KUKA KRL program: S_11_pc_at_cell_01.src, S_11_pc_at_cell_01.dat

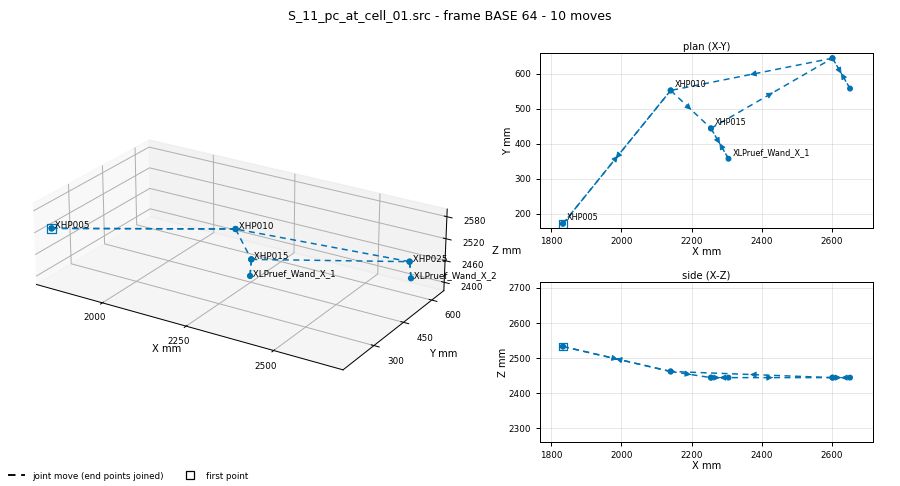
[picture p0: tool path of S_11_pc_at_cell_01.src in frame BASE 64, 10 of 12 moves have a stored position in this frame; points joined in program order, loops and branches not executed]
--- S_11_pc_at_cell_01.src ---
&ACCESS RVP
&REL 9
&COMMENT DAI_H_SOP_pc_at_cell_01
&PARAM EDITMASK = DAI
&PARAM TEMPLATE = C:\KRC\roboter\template\vg_appl
&PARAM DISKPATH = KRC:\R1\H_Prog\DAI_SOP
DEF S_11_pc_at_cell_01( )
;FOLD INI;%{PE}
  ;FOLD BASISTECH INI
    GLOBAL INTERRUPT DECL 3 WHEN $STOPMESS==TRUE DO IR_STOPM ( )
    INTERRUPT ON 3
    BAS (#INITMOV,0 )
  ;ENDFOLD (BASISTECH INI)
  ;FOLD USER INI
    ;Make your modifications here
  ;ENDFOLD (USER INI)
;ENDFOLD (INI)
;FOLD ; Anlagenbezeichn: HC53_C    Stations-Nr: 060RB_100;%{PE}
;FOLD Parameters ;%{h}
;Params IlfProvider=kukaroboter.basistech.inlineforms.comments.comment; Kuka.Content=Anlagenbezeichn: HC53_C    Stations-Nr: 060RB_100
;ENDFOLD
;ENDFOLD
;FOLD ; Stand / Version: V1.0;%{PE}
;FOLD Parameters ;%{h}
;Params IlfProvider=kukaroboter.basistech.inlineforms.comments.comment; Kuka.Content=Stand / Version: V1.0
;ENDFOLD
;ENDFOLD
;FOLD ; Name Bearbeiter: EBZ-AE;%{PE}
;FOLD Parameters ;%{h}
;Params IlfProvider=kukaroboter.basistech.inlineforms.comments.comment; Kuka.Content=Name Bearbeiter: EBZ-AE
;ENDFOLD
;ENDFOLD
;FOLD ; Translator Version:29.01.2024 - Version 15.08;%{PE}
;FOLD Parameters ;%{h}
;Params IlfProvider=kukaroboter.basistech.inlineforms.comments.comment; Kuka.Content=Translator Version:29.01.2024 - Version 15.08
;ENDFOLD
;ENDFOLD

REPEAT

;FOLD MSG_T1
MSG_SHOW("DAI_H_SOP",#quit,999,"dai_h_sop_ok_0")
;ENDFOLD

; ***************************************
; A C H T U N G !!! Nur in $T1 abfahren
; ***************************************
UNTIL $T1 == TRUE

; ***************************************
; Pruefende Waende = 2
;----------------------------------------
; Lademagazin in undefinierte
; Position verfahren, damit Raum
; aktiviert wird.
;FOLD WAIT FOR ( IN 1026 'Vordefinierter Eingang immer ruckgesetzt.' )  ;%{PE}
;FOLD Parameters ;%{h}
;Params IlfProvider=kukaroboter.basistech.inlineforms.logics.waitfor; Kuka.WaitLogicTerm1=None; Kuka.WaitForNot1=False; Kuka.WaitLogicOp2.Term1=None; Kuka.WaitForNot2.Term1=False; Kuka.WaitForSysVar2.Term1=IN; Kuka.WaitForIndex2.Term1=1026; Kuka.WaitForIndexName2.Term1=Vordefinierter Eingang immer ruckgesetzt.; Kuka.WaitForTermNumbers=1; Kuka.WaitForOpNumbers=2; Kuka.WaitForCont=False
;ENDFOLD
WAIT FOR  ( $IN[1026] )
;ENDFOLD
; ***************************************

;FOLD PTP HOME Vel=100 % DEFAULT;%{PE}
;FOLD Parameters ;%{h}
;Params IlfProvider=kukaroboter.basistech.inlineforms.movement.old; Kuka.IsGlobalPoint=False; Kuka.PointName=HOME; Kuka.BlendingEnabled=False; Kuka.MoveDataPtpName=DEFAULT; Kuka.VelocityPtp=100; Kuka.CurrentCDSetIndex=0; Kuka.MovementParameterFieldEnabled=True; IlfCommand=PTP
;ENDFOLD
$BWDSTART = FALSE
PDAT_ACT = PDEFAULT
FDAT_ACT = FHOME
BAS(#PTP_PARAMS, 100.0)
SET_CD_PARAMS (0)
PTP XHOME
;ENDFOLD

;Dynamische Pruefung Teil vorhanden
;FOLD PartPresent.CheckOff #1:5277, #2:5278, #3:1025, #4:1025, #5:1025, #6:1025, Bounce Time:100, Constant: Yes;%{PE}%
CheckPartPresent(5277,5278,1025,1025,1025,1025,100, True,FALSE)
;ENDFOLD

;Greifer-Ventile betatigen/pruefen
;FOLD DAI_GripValveCheck.Valve2 State:Fixierstift Ausfahren Gs, 060GRH101-QM1;%{PE}%
CheckValveState(2,1)
;ENDFOLD
;FOLD DAI_GripValveCheck.Valve3 State:Spanner Oeffnen Gs, 060GRH101-QM2;%{PE}%
CheckValveState(3,1)
;ENDFOLD
;FOLD DAI_GripValveCheck.Valve4 State:Spanner Oeffnen Gs, 060GRH101-QM3;%{PE}%
CheckValveState(4,1)
;ENDFOLD

;FOLD PTP HP005 Vel=100 % PDAT2 Tool[64]:Zero Base[64]:Zero;%{PE}
;FOLD Parameters ;%{h}
;Params IlfProvider=kukaroboter.basistech.inlineforms.movement.old; Kuka.IsGlobalPoint=False; Kuka.PointName=HP005; Kuka.BlendingEnabled=False; Kuka.MoveDataPtpName=PDAT2; Kuka.VelocityPtp=100; Kuka.CurrentCDSetIndex=0; Kuka.MovementParameterFieldEnabled=True; IlfCommand=PTP
;ENDFOLD
$BWDSTART = FALSE
PDAT_ACT = PPDAT2
FDAT_ACT = FHP005
BAS(#PTP_PARAMS, 100.0)
SET_CD_PARAMS (0)
PTP XHP005
;ENDFOLD
;FOLD PTP HP010 Vel=100 % PDAT3 Tool[64]:Zero Base[64]:Zero;%{PE}
;FOLD Parameters ;%{h}
;Params IlfProvider=kukaroboter.basistech.inlineforms.movement.old; Kuka.IsGlobalPoint=False; Kuka.PointName=HP010; Kuka.BlendingEnabled=False; Kuka.MoveDataPtpName=PDAT3; Kuka.VelocityPtp=100; Kuka.CurrentCDSetIndex=0; Kuka.MovementParameterFieldEnabled=True; IlfCommand=PTP
;ENDFOLD
$BWDSTART = FALSE
PDAT_ACT = PPDAT3
FDAT_ACT = FHP010
BAS(#PTP_PARAMS, 100.0)
SET_CD_PARAMS (0)
PTP XHP010
;ENDFOLD
;FOLD PTP HP015 Vel=100 % PDAT4 Tool[64]:Zero Base[64]:Zero;%{PE}
;FOLD Parameters ;%{h}
;Params IlfProvider=kukaroboter.basistech.inlineforms.movement.old; Kuka.IsGlobalPoint=False; Kuka.PointName=HP015; Kuka.BlendingEnabled=False; Kuka.MoveDataPtpName=PDAT4; Kuka.VelocityPtp=100; Kuka.CurrentCDSetIndex=0; Kuka.MovementParameterFieldEnabled=True; IlfCommand=PTP
;ENDFOLD
$BWDSTART = FALSE
PDAT_ACT = PPDAT4
FDAT_ACT = FHP015
BAS(#PTP_PARAMS, 100.0)
SET_CD_PARAMS (0)
PTP XHP015
;ENDFOLD

; Pruefung Flache 1 erste Position
;FOLD PTP LPruef_Wand_X_1 Vel=100 % PDAT04 Tool[64]:Zero Base[64]:Zero ;%{PE}
;FOLD Parameters ;%{h}
;Params IlfProvider=kukaroboter.basistech.inlineforms.movement.old; Kuka.IsGlobalPoint=False; Kuka.PointName=LPruef_Wand_X_1; Kuka.BlendingEnabled=False; Kuka.MoveDataPtpName=PDAT04; Kuka.VelocityPtp=100; Kuka.CurrentCDSetIndex=0; Kuka.MovementParameterFieldEnabled=True; IlfCommand=PTP
;ENDFOLD
$BWDSTART = FALSE
PDAT_ACT = PPDAT04
FDAT_ACT = FLPruef_Wand_X_1
BAS(#PTP_PARAMS, 100.0)
SET_CD_PARAMS (0)
PTP XLPruef_Wand_X_1
;ENDFOLD

;FOLD PTP HP020 Vel=100 % PDAT03 Tool[64]:Zero Base[64]:Zero ;%{PE}
;FOLD Parameters ;%{h}
;Params IlfProvider=kukaroboter.basistech.inlineforms.movement.old; Kuka.IsGlobalPoint=False; Kuka.PointName=HP020; Kuka.BlendingEnabled=False; Kuka.MoveDataPtpName=PDAT03; Kuka.VelocityPtp=100; Kuka.CurrentCDSetIndex=0; Kuka.MovementParameterFieldEnabled=True; IlfCommand=PTP
;ENDFOLD
$BWDSTART = FALSE
PDAT_ACT = PPDAT03
FDAT_ACT = FHP020
BAS(#PTP_PARAMS, 100.0)
SET_CD_PARAMS (0)
PTP XHP020
;ENDFOLD

;FOLD PTP HP025 Vel=100 % PDAT7 Tool[64]:Zero Base[64]:Zero;%{PE}
;FOLD Parameters ;%{h}
;Params IlfProvider=kukaroboter.basistech.inlineforms.movement.old; Kuka.IsGlobalPoint=False; Kuka.PointName=HP025; Kuka.BlendingEnabled=False; Kuka.MoveDataPtpName=PDAT7; Kuka.VelocityPtp=100; Kuka.CurrentCDSetIndex=0; Kuka.MovementParameterFieldEnabled=True; IlfCommand=PTP
;ENDFOLD
$BWDSTART = FALSE
PDAT_ACT = PPDAT7
FDAT_ACT = FHP025
BAS(#PTP_PARAMS, 100.0)
SET_CD_PARAMS (0)
PTP XHP025
;ENDFOLD

; Pruefung Flache 1 zweite Position
;FOLD PTP LPruef_Wand_X_2 Vel=100 % PDAT02 Tool[64]:Zero Base[64]:Zero ;%{PE}
;FOLD Parameters ;%{h}
;Params IlfProvider=kukaroboter.basistech.inlineforms.movement.old; Kuka.IsGlobalPoint=False; Kuka.PointName=LPruef_Wand_X_2; Kuka.BlendingEnabled=False; Kuka.MoveDataPtpName=PDAT02; Kuka.VelocityPtp=100; Kuka.CurrentCDSetIndex=0; Kuka.MovementParameterFieldEnabled=True; IlfCommand=PTP
;ENDFOLD
$BWDSTART = FALSE
PDAT_ACT = PPDAT02
FDAT_ACT = FLPruef_Wand_X_2
BAS(#PTP_PARAMS, 100.0)
SET_CD_PARAMS (0)
PTP XLPruef_Wand_X_2
;ENDFOLD

;FOLD PTP HP030 Vel=100 % PDAT01 Tool[64]:Zero Base[64]:Zero ;%{PE}
;FOLD Parameters ;%{h}
;Params IlfProvider=kukaroboter.basistech.inlineforms.movement.old; Kuka.IsGlobalPoint=False; Kuka.PointName=HP030; Kuka.BlendingEnabled=False; Kuka.MoveDataPtpName=PDAT01; Kuka.VelocityPtp=100; Kuka.CurrentCDSetIndex=0; Kuka.MovementParameterFieldEnabled=True; IlfCommand=PTP
;ENDFOLD
$BWDSTART = FALSE
PDAT_ACT = PPDAT01
FDAT_ACT = FHP030
BAS(#PTP_PARAMS, 100.0)
SET_CD_PARAMS (0)
PTP XHP030
;ENDFOLD

;FOLD PTP HP040 Vel=100 % PDAT05 Tool[64]:Zero Base[64]:Zero ;%{PE}
;FOLD Parameters ;%{h}
;Params IlfProvider=kukaroboter.basistech.inlineforms.movement.old; Kuka.IsGlobalPoint=False; Kuka.PointName=HP040; Kuka.BlendingEnabled=False; Kuka.MoveDataPtpName=PDAT05; Kuka.VelocityPtp=100; Kuka.CurrentCDSetIndex=0; Kuka.MovementParameterFieldEnabled=True; IlfCommand=PTP
;ENDFOLD
$BWDSTART = FALSE
PDAT_ACT = PPDAT05
FDAT_ACT = FHP040
BAS(#PTP_PARAMS, 100.0)
SET_CD_PARAMS (0)
PTP XHP040
;ENDFOLD
;FOLD PTP HP045 Vel=100 % PDAT13 Tool[64]:Zero Base[64]:Zero;%{PE}
;FOLD Parameters ;%{h}
;Params IlfProvider=kukaroboter.basistech.inlineforms.movement.old; Kuka.IsGlobalPoint=False; Kuka.PointName=HP045; Kuka.BlendingEnabled=False; Kuka.MoveDataPtpName=PDAT13; Kuka.VelocityPtp=100; Kuka.CurrentCDSetIndex=0; Kuka.MovementParameterFieldEnabled=True; IlfCommand=PTP
;ENDFOLD
$BWDSTART = FALSE
PDAT_ACT = PPDAT13
FDAT_ACT = FHP045
BAS(#PTP_PARAMS, 100.0)
SET_CD_PARAMS (0)
PTP XHP045
;ENDFOLD

;FOLD PTP HOME Vel=100 % DEFAULT;%{PE}
;FOLD Parameters ;%{h}
;Params IlfProvider=kukaroboter.basistech.inlineforms.movement.old; Kuka.IsGlobalPoint=False; Kuka.PointName=HOME; Kuka.BlendingEnabled=False; Kuka.MoveDataPtpName=DEFAULT; Kuka.VelocityPtp=100; Kuka.CurrentCDSetIndex=0; Kuka.MovementParameterFieldEnabled=True; IlfCommand=PTP
;ENDFOLD
$BWDSTART = FALSE
PDAT_ACT = PDEFAULT
FDAT_ACT = FHOME
BAS(#PTP_PARAMS, 100.0)
SET_CD_PARAMS (0)
PTP XHOME
;ENDFOLD

;----------------------------------------
; Lademagazin schliessen und
; und Quittieren.
;FOLD WAIT FOR ( IN 1026 'Vordefinierter Eingang immer ruckgesetzt.' )  ;%{PE}
;FOLD Parameters ;%{h}
;Params IlfProvider=kukaroboter.basistech.inlineforms.logics.waitfor; Kuka.WaitLogicTerm1=None; Kuka.WaitForNot1=False; Kuka.WaitLogicOp2.Term1=None; Kuka.WaitForNot2.Term1=False; Kuka.WaitForSysVar2.Term1=IN; Kuka.WaitForIndex2.Term1=1026; Kuka.WaitForIndexName2.Term1=Vordefinierter Eingang immer ruckgesetzt.; Kuka.WaitForTermNumbers=1; Kuka.WaitForOpNumbers=2; Kuka.WaitForCont=False
;ENDFOLD
WAIT FOR  ( $IN[1026] )
;ENDFOLD
; ***************************************
 ;Collision detection - Off
;FOLD COLLDETECT Off ;%{PE}
;FOLD Parameters ;%{h}
;Params IlfProvider=kukaroboter.basistech.inlineforms.colldetect.off; CollDetect.Command=Off
;ENDFOLD
USE_CD_PARAMS(0)
;ENDFOLD
END

--- S_11_pc_at_cell_01.dat ---
&ACCESS RVP
&REL 11
&COMMENT DAI_H_SOP_pc_at_cell_01
&PARAM EDITMASK = DAI
&PARAM TEMPLATE = C:\KRC\roboter\template\vg_appl
&PARAM DISKPATH = KRC:\R1\H_Prog\DAI_SOP
DEFDAT  S_11_PC_AT_CELL_01
;FOLD EXTERNAL DECLARATIONS;%{PE}%MKUKATPBASIS,%CEXT,%VCOMMON,%P
;FOLD BASISTECH EXT;%{PE}%MKUKATPBASIS,%CEXT,%VEXT,%P
EXT  BAS (BAS_COMMAND  :IN,REAL  :IN )
DECL INT SUCCESS
;ENDFOLD (BASISTECH EXT)
;FOLD USER EXT;%{E}%MKUKATPUSER,%CEXT,%VEXT,%P
;Make your modifications here
;ENDFOLD (USER EXT)
;FOLD COLLISION
EXT  COLLSTOP (INT  :IN,INT  :IN )
;ENDFOLD  (Collision)
;ENDFOLD (EXTERNAL DECLERATIONS)
DECL BASIS_SUGG_T LAST_BASIS={POINT1[] "P0                      ",POINT2[] "P0                      ",CP_PARAMS[] "CPDAT0                  ",PTP_PARAMS[] "PDAT0                   ",CONT[] "                        ",CP_VEL[] "2.0                     ",PTP_VEL[] "100                     ",SYNC_PARAMS[] "SYNCDAT                 ",SPL_NAME[] "S0                      ",A_PARAMS[] "ADAT0                   "}
DECL FDAT FHOME={TOOL_NO 64,BASE_NO 64,IPO_FRAME #BASE,POINT2[] " "}
DECL PDAT PPDAT1={VEL 100.000,ACC 100.000,APO_DIST 0.0,APO_MODE #CDIS,GEAR_JERK 50.0000,EXAX_IGN 0}
DECL E6POS XHP005={X 1833.41858,Y 172.027740,Z 2533.01074,A -100.250282,B -31.8846416,C -108.130798,S 18,T 3,E1 -846.026428,E2 0.0,E3 0.0,E4 0.0,E5 0.0,E6 0.0}
DECL FDAT FHP005={TOOL_NO 64,BASE_NO 64,IPO_FRAME #BASE,POINT2[] " "}
DECL PDAT PPDAT2={VEL 100.000,ACC 100.000,APO_DIST 0.0,APO_MODE #CDIS,GEAR_JERK 50.0000,EXAX_IGN 0}
DECL E6POS XHP010={X 2140.48633,Y 551.821594,Z 2461.88916,A 140.541840,B -65.4589691,C 22.4935665,S 18,T 3,E1 -1300.00,E2 0.0,E3 0.0,E4 0.0,E5 0.0,E6 0.0}
DECL FDAT FHP010={TOOL_NO 64,BASE_NO 64,IPO_FRAME #BASE,POINT2[] " "}
DECL PDAT PPDAT3={VEL 100.000,ACC 100.000,APO_DIST 0.0,APO_MODE #CDIS,GEAR_JERK 50.0000,EXAX_IGN 0}
DECL E6POS XHP015={X 2255.26440,Y 443.720276,Z 2444.36743,A 127.156387,B -65.5106659,C 27.3130951,S 18,T 3,E1 -1300.00,E2 0.0,E3 0.0,E4 0.0,E5 0.0,E6 0.0}
DECL FDAT FHP015={TOOL_NO 64,BASE_NO 64,IPO_FRAME #BASE,POINT2[] " "}
DECL PDAT PPDAT4={VEL 100.000,ACC 100.000,APO_DIST 0.0,APO_MODE #CDIS,GEAR_JERK 50.0000,EXAX_IGN 0}
DECL E6POS XLPruef_Wand_X_1={X 2305.27026,Y 357.121216,Z 2444.37134,A 127.156921,B -65.5106735,C 27.3124809,S 18,T 3,E1 -1300.00,E2 0.0,E3 0.0,E4 0.0,E5 0.0,E6 0.0}
DECL FDAT FLPruef_Wand_X_1={TOOL_NO 64,BASE_NO 64,IPO_FRAME #BASE,POINT2[] " "}
DECL LDAT LCPDAT5={VEL 0.500000,ACC 100.000,APO_DIST 0.0,APO_FAC 50.0000,AXIS_VEL 100.000,AXIS_ACC 100.000,ORI_TYP #VAR,CIRC_TYP #BASE,JERK_FAC 50.0000,GEAR_JERK 50.0000,EXAX_IGN 0}
DECL E6POS XHP020={X 2255.27417,Y 443.726715,Z 2444.37134,A 127.156418,B -65.5106735,C 27.3130760,S 18,T 3,E1 -1300.00,E2 0.0,E3 0.0,E4 0.0,E5 0.0,E6 0.0}
DECL FDAT FHP020={TOOL_NO 64,BASE_NO 64,IPO_FRAME #BASE,POINT2[] " "}
DECL LDAT LCPDAT6={VEL 0.500000,ACC 100.000,APO_DIST 0.0,APO_FAC 50.0000,AXIS_VEL 100.000,AXIS_ACC 100.000,ORI_TYP #VAR,CIRC_TYP #BASE,JERK_FAC 50.0000,GEAR_JERK 50.0000,EXAX_IGN 0}
DECL E6POS XHP025={X 2601.67798,Y 643.723938,Z 2444.36621,A 127.156319,B -65.5106125,C 27.3132076,S 18,T 3,E1 -1300.00,E2 0.0,E3 0.0,E4 0.0,E5 0.0,E6 0.0}
DECL FDAT FHP025={TOOL_NO 64,BASE_NO 64,IPO_FRAME #BASE,POINT2[] " "}
DECL PDAT PPDAT7={VEL 100.000,ACC 100.000,APO_DIST 0.0,APO_MODE #CDIS,GEAR_JERK 50.0000,EXAX_IGN 0}
DECL E6POS XLPruef_Wand_X_2={X 2651.68066,Y 557.123108,Z 2444.36597,A 127.156326,B -65.5106201,C 27.3131962,S 18,T 3,E1 -1300.00,E2 0.0,E3 0.0,E4 0.0,E5 0.0,E6 0.0}
DECL FDAT FLPruef_Wand_X_2={TOOL_NO 64,BASE_NO 64,IPO_FRAME #BASE,POINT2[] " "}
DECL LDAT LCPDAT8={VEL 0.500000,ACC 100.000,APO_DIST 0.0,APO_FAC 50.0000,AXIS_VEL 100.000,AXIS_ACC 100.000,ORI_TYP #VAR,CIRC_TYP #BASE,JERK_FAC 50.0000,GEAR_JERK 50.0000,EXAX_IGN 0}
DECL E6POS XHP030={X 2601.68433,Y 643.728271,Z 2444.36523,A 127.156342,B -65.5106201,C 27.3131847,S 18,T 3,E1 -1300.00,E2 0.0,E3 0.0,E4 0.0,E5 0.0,E6 0.0}
DECL FDAT FHP030={TOOL_NO 64,BASE_NO 64,IPO_FRAME #BASE,POINT2[] " "}
DECL LDAT LCPDAT9={VEL 0.500000,ACC 100.000,APO_DIST 0.0,APO_FAC 50.0000,AXIS_VEL 100.000,AXIS_ACC 100.000,ORI_TYP #VAR,CIRC_TYP #BASE,JERK_FAC 50.0000,GEAR_JERK 50.0000,EXAX_IGN 0}
DECL E6POS XHP035={X 2651.62183,Y 672.557,Z 3077.02612,A -175.231079,B -15.2318830,C -47.7739716,S 18,T 3,E1 -1300.00,E2 0.0,E3 0.0,E4 0.0,E5 0.0,E6 0.0}
DECL FDAT FHP035={TOOL_NO 64,BASE_NO 64,IPO_FRAME #BASE,POINT2[] " "}
DECL PDAT PPDAT10={VEL 100.000,ACC 100.000,APO_DIST 0.0,APO_MODE #CDIS,GEAR_JERK 50.0000,EXAX_IGN 0}
DECL E6POS XLPruef_Wand_X_3={X 2701.62817,Y 585.958252,Z 3077.02954,A -175.231064,B -15.2318983,C -47.7739716,S 18,T 3,E1 -1300.00,E2 0.0,E3 0.0,E4 0.0,E5 0.0,E6 0.0}
DECL FDAT FLPruef_Wand_X_3={TOOL_NO 64,BASE_NO 64,IPO_FRAME #BASE,POINT2[] " "}
DECL LDAT LCPDAT11={VEL 0.500000,ACC 100.000,APO_DIST 0.0,APO_FAC 50.0000,AXIS_VEL 100.000,AXIS_ACC 100.000,ORI_TYP #VAR,CIRC_TYP #BASE,JERK_FAC 50.0000,GEAR_JERK 50.0000,EXAX_IGN 0}
DECL E6POS XHP040={X 2140.48657,Y 551.821777,Z 2461.88867,A 140.541809,B -65.4589691,C 22.4935913,S 18,T 3,E1 -1300.00,E2 0.0,E3 0.0,E4 0.0,E5 0.0,E6 0.0}
DECL FDAT FHP040={TOOL_NO 64,BASE_NO 64,IPO_FRAME #BASE,POINT2[] " "}
DECL LDAT LCPDAT12={VEL 0.500000,ACC 100.000,APO_DIST 0.0,APO_FAC 50.0000,AXIS_VEL 100.000,AXIS_ACC 100.000,ORI_TYP #VAR,CIRC_TYP #BASE,JERK_FAC 50.0000,GEAR_JERK 50.0000,EXAX_IGN 0}
DECL E6POS XHP045={X 1833.41895,Y 172.028259,Z 2533.01,A -100.250282,B -31.8846664,C -108.130821,S 18,T 3,E1 -846.026428,E2 0.0,E3 0.0,E4 0.0,E5 0.0,E6 0.0}
DECL FDAT FHP045={TOOL_NO 64,BASE_NO 64,IPO_FRAME #BASE,POINT2[] " "}
DECL PDAT PPDAT13={VEL 100.000,ACC 100.000,APO_DIST 0.0,APO_MODE #CDIS,GEAR_JERK 50.0000,EXAX_IGN 0}
DECL PDAT PPDAT14={VEL 100.000,ACC 100.000,APO_DIST 0.0,APO_MODE #CDIS,GEAR_JERK 50.0000,EXAX_IGN 0}
DECL PDAT PPDAT01={VEL 100.000,ACC 100.000,APO_DIST 500.000,APO_MODE #CDIS,GEAR_JERK 100.000,EXAX_IGN 0}
DECL MODULEPARAM_T LAST_TP_PARAMS={PARAMS[] "Kuka.PointName=HP040; Kuka.FrameData.base_no=64; Kuka.FrameData.tool_no=64; Kuka.FrameData.ipo_frame=#BASE; Kuka.FrameData.point2=; Kuka.isglobalpoint=False; Kuka.MoveDataPtpName=PDAT05; Kuka.MovementDataPdat.apo_mode=#CDIS; Kuka.MovementDataPdat.apo_dist=500; Kuka.MovementData.vel=100; Kuka.MovementData.acc=100; Kuka.MovementData.exax_ign=0; Kuka.VelocityPtp=100; Kuka.BlendingEnabled=False; Kuka.APXEnabled=False; Kuka.CurrentCDSetIndex=0          "}
DECL PDAT PPDAT02={VEL 100.000,ACC 100.000,APO_DIST 500.000,APO_MODE #CDIS,GEAR_JERK 100.000,EXAX_IGN 0}
DECL PDAT PPDAT03={VEL 100.000,ACC 100.000,APO_DIST 500.000,APO_MODE #CDIS,GEAR_JERK 100.000,EXAX_IGN 0}
DECL PDAT PPDAT04={VEL 100.000,ACC 100.000,APO_DIST 500.000,APO_MODE #CDIS,GEAR_JERK 100.000,EXAX_IGN 0}
DECL PDAT PPDAT05={VEL 100.000,ACC 100.000,APO_DIST 500.000,APO_MODE #CDIS,GEAR_JERK 100.000,EXAX_IGN 0}
ENDDAT
